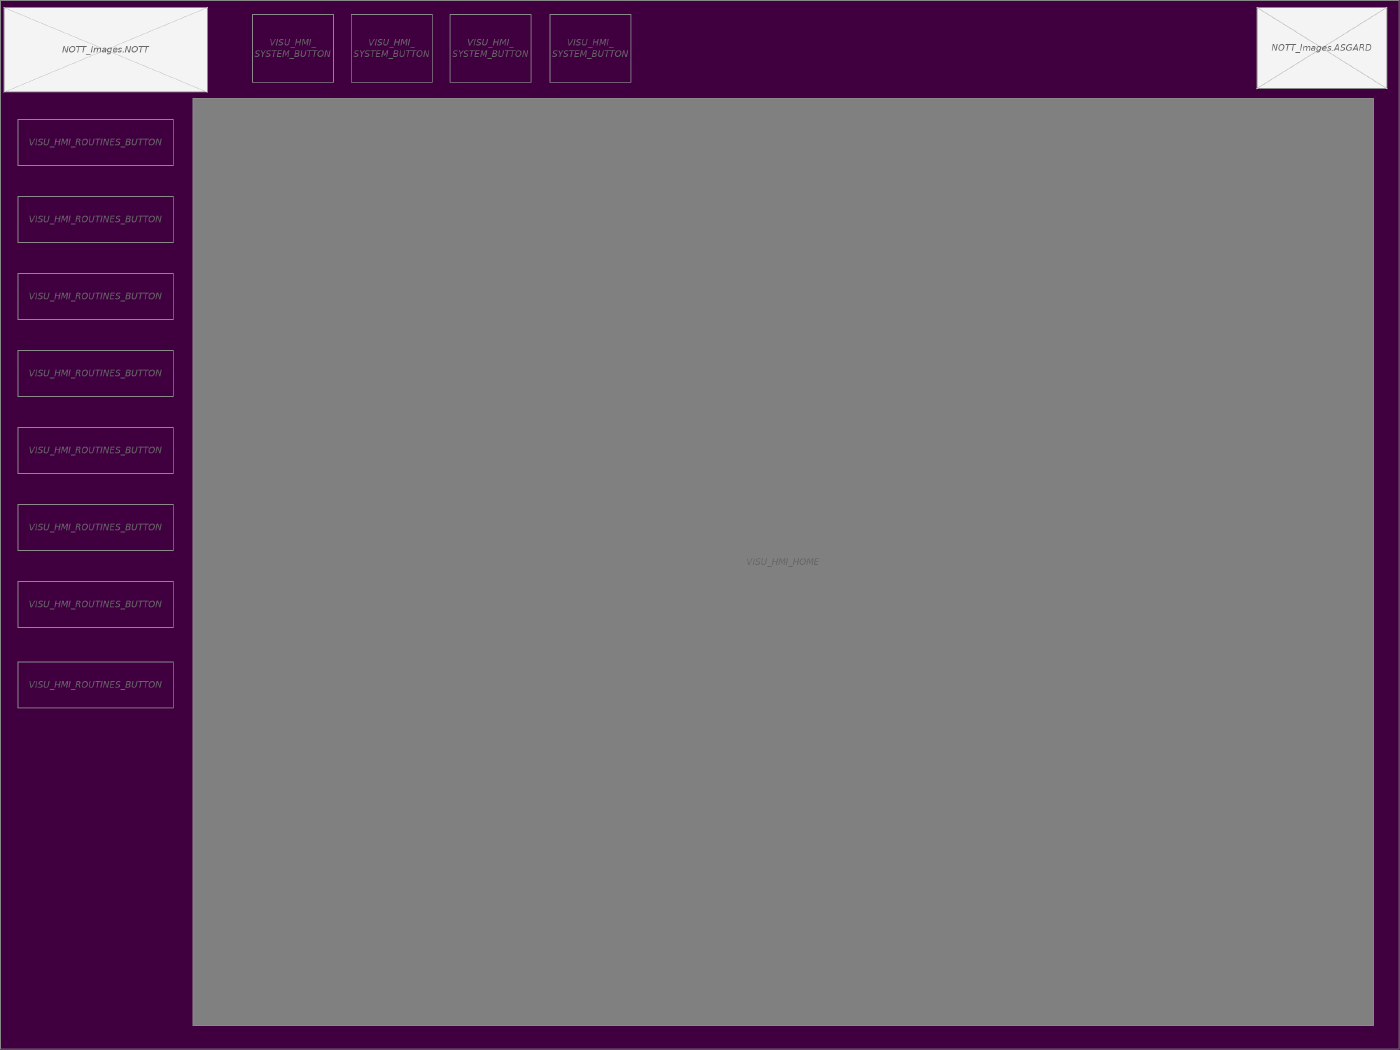
VISUALIZATION VISU_HMI  // 1600x1200
    Rectangle (220,112 1350x1060)
    Frame (220,112 1350x1060), frame switch variable: PRG_HMI.eActiveTab
        shows VISU_HMI_HOME(m_instance := MAIN.nott_ics)
        shows VISU_HMI_SERVICES(m_Instance := MAIN.fbServices)
        shows VISU_HMI_EVENTS()
        shows VISU_HMI_CRYO_INTERLOCKS()
        shows VISU_HMI_SHUTTERS()
        shows VISU_HMI_TIP_TILT(m_Hmi := PRG_HMI.fbTipTilt)
        shows VISU_HMI_DELAY_LINES()
        shows VISU_HMI_CO2_TRANS_STAGES()
        shows VISU_HMI_ZNSE_ACTUATORS()
        shows VISU_HMI_BIREFRINGENCE()
        shows VISU_HMI_BEAM_SPLITTER()
        shows VISU_HMI_CO2_PRESSURE()
        shows VISU_HMI_CRY(met_cryo_ctrl := MAIN.met_cryo_ctrl, m_Hmi := PRG_HMI.fbCry)
        shows VISU_HMI_CFO()
        shows VISU_HMI_IMG(m_Temperatures := MAIN.met_cryo_ctrl.met_temp, m_Voters := MAIN.met_cryo_ctrl.met_voters, m_Tctrl := MAIN.met_cryo_ctrl.met_tctrl, m_Heaters := MAIN.met_cryo_ctrl.met_heaters, m_Lakeshores := MAIN.met_cryo_ctrl.met_lakeshores, m_Hmi := PRG_HMI.fbImg)
        shows VISU_HMI_LMS()
        shows VISU_HMI_SCA(m_Temperatures := MAIN.met_cryo_ctrl.met_temp, m_Voters := MAIN.met_cryo_ctrl.met_voters, m_Tctrl := MAIN.met_cryo_ctrl.met_tctrl, m_Heaters := MAIN.met_cryo_ctrl.met_heaters, m_Lakeshores := MAIN.met_cryo_ctrl.met_lakeshores, m_Hmi := PRG_HMI.fbSca)
        shows VISU_HMI_HEATERS()
        shows VISU_HMI_EVENTS()
        shows VISU_HMI_PRESSURES()
        shows VISU_HMI_COOLERS()
        shows VISU_HMI_PUMPS(m_Hmi := PRG_HMI.fbPumps)
        shows VISU_HMI_TEMPERATURES(met_cryo_ctrl := MAIN.met_cryo_ctrl, m_Hmi := PRG_HMI.fbTemperatures)
        shows VISU_HMI_ICS_INTERLOCKS()
        shows VISU_HMI_DETECTORS()
        shows VISU_HMI_CONTROL_LOOPS()
        p1199675002: PRG_HMI.fbSca
        p1171169602: PRG_HMI.fbPumps
    Frame (288,16 93x78)
        shows VISU_HMI_SYSTEM_BUTTON(m_Hmi := PRG_HMI.fbHomeButton)
        OnMouseClick: execute { PRG_HMI.eActiveTab := E_HMI_TABS.HOME; }
    Frame (401,16 93x78)
        shows VISU_HMI_SYSTEM_BUTTON(m_Hmi := PRG_HMI.fbServicesButton)
        OnMouseClick: execute { PRG_HMI.eActiveTab := E_HMI_TABS.SERVICES; }
    Frame (514,16 93x78)
        shows VISU_HMI_SYSTEM_BUTTON(m_Hmi := PRG_HMI.fbEventsButton)
        OnMouseClick: execute { PRG_HMI.eActiveTab := E_HMI_TABS.EVENTS; }
    Frame (628,16 93x78)
        shows VISU_HMI_SYSTEM_BUTTON(m_Hmi := PRG_HMI.fbCryoInterlocksButton)
        OnMouseClick: execute { PRG_HMI.eActiveTab := E_HMI_TABS.CRYO_INTERLOCKS; }
    Frame (20,136 178x53)
        shows VISU_HMI_ROUTINES_BUTTON(m_Hmi := PRG_HMI.fbShuttersButton)
        OnMouseClick: execute { PRG_HMI.eActiveTab := E_HMI_TABS.SHUTTERS; }
    Frame (20,224 178x53)
        shows VISU_HMI_ROUTINES_BUTTON(m_Hmi := PRG_HMI.fbTipTiltButton)
        OnMouseClick: execute { PRG_HMI.eActiveTab := E_HMI_TABS.TIP_TILT; }
    Frame (20,312 178x53)
        shows VISU_HMI_ROUTINES_BUTTON(m_Hmi := PRG_HMI.fbDelayLinesButton)
        OnMouseClick: execute { PRG_HMI.eActiveTab := E_HMI_TABS.DELAY_LINES; }
    Frame (20,400 178x53)
        shows VISU_HMI_ROUTINES_BUTTON(m_Hmi := PRG_HMI.fbCO2TransStagesButton)
        OnMouseClick: execute { PRG_HMI.eActiveTab := E_HMI_TABS.CO2_TRANSLATION_STAGES; }
    Frame (20,488 178x53)
        shows VISU_HMI_ROUTINES_BUTTON(m_Hmi := PRG_HMI.fbZnSeActuatorsButton)
        OnMouseClick: execute { PRG_HMI.eActiveTab := E_HMI_TABS.ZNSE_ACTUATORS; }
    Frame (20,576 178x53)
        shows VISU_HMI_ROUTINES_BUTTON(m_Hmi := PRG_HMI.fbBirefringenceButton)
        OnMouseClick: execute { PRG_HMI.eActiveTab := E_HMI_TABS.BIREFRINGENCE_ACTUATORS; }
    Frame (20,664 178x53)
        shows VISU_HMI_ROUTINES_BUTTON(m_Hmi := PRG_HMI.fbBeamSplitterButton)
        OnMouseClick: execute { PRG_HMI.eActiveTab := E_HMI_TABS.CALIBRATION_UNIT_BEAM_SPLITER; }
    Frame (20,756 178x53)
        shows VISU_HMI_ROUTINES_BUTTON(m_Hmi := PRG_HMI.fbCO2PressureButton)
        OnMouseClick: execute { PRG_HMI.eActiveTab := E_HMI_TABS.CO2_PRESSURE_CONTROL; }
    Image (4,8 233x97), image: NOTT_Images.NOTT
    Image (1436,8 149x93), image: NOTT_Images.ASGARD
END_VISUALIZATION

(* stored: Version 1.1.0.1, ProductVersion 3.1.4024.15
   Visu VISU_HMI: Id {014faa3a-f820-47de-a8b1-8bb3f9189724} *)
